PROGRAM MOVMENT_Controller
VAR
	X_Axis:				FB_PTP_AXIS_ABS_CONTROL;
	Y_Axis:				FB_PTP_AXIS_ABS_CONTROL;
	Z_Axis:				FB_PTP_AXIS_ABS_CONTROL;
	
	eJogMode: 				E_JogMode;
END_VAR

IF (G_sControl.ManualMoveMode) THEN
	eJogMode:= MC_JOGMODE_CONTINOUS;
ELSE
	eJogMode:= MC_JOGMODE_INCHING;
END_IF

ACT_AXIS_CTRL();

ACTION ACT_AXIS_CTRL:
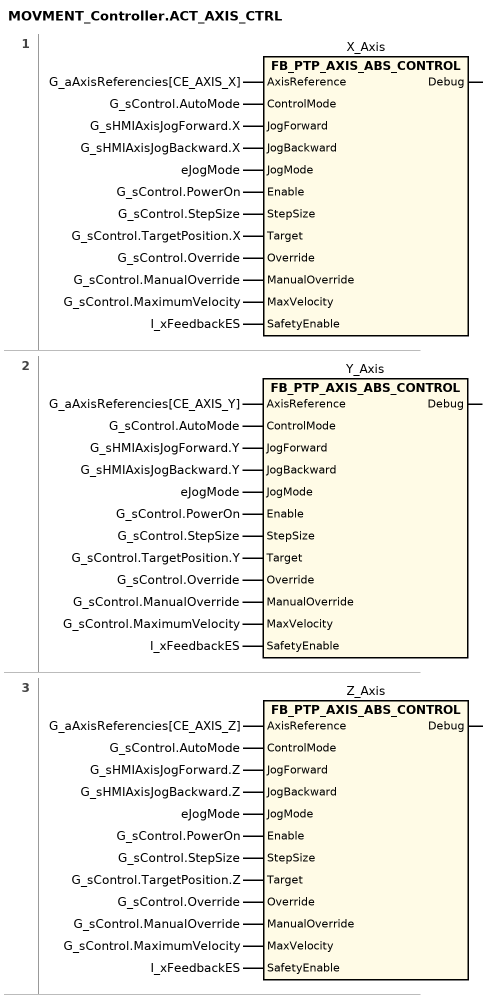
// NETWORK 1
X_Axis(
    AxisReference := G_aAxisReferencies[CE_AXIS_X],
    ControlMode := G_sControl.AutoMode,
    JogForward := G_sHMIAxisJogForward.X,
    JogBackward := G_sHMIAxisJogBackward.X,
    JogMode := eJogMode,
    Enable := G_sControl.PowerOn,
    StepSize := G_sControl.StepSize,
    Target := G_sControl.TargetPosition.X,
    Override := G_sControl.Override,
    ManualOverride := G_sControl.ManualOverride,
    MaxVelocity := G_sControl.MaximumVelocity,
    SafetyEnable := I_xFeedbackES); // FB_PTP_AXIS_ABS_CONTROL

// NETWORK 2
Y_Axis(
    AxisReference := G_aAxisReferencies[CE_AXIS_Y],
    ControlMode := G_sControl.AutoMode,
    JogForward := G_sHMIAxisJogForward.Y,
    JogBackward := G_sHMIAxisJogBackward.Y,
    JogMode := eJogMode,
    Enable := G_sControl.PowerOn,
    StepSize := G_sControl.StepSize,
    Target := G_sControl.TargetPosition.Y,
    Override := G_sControl.Override,
    ManualOverride := G_sControl.ManualOverride,
    MaxVelocity := G_sControl.MaximumVelocity,
    SafetyEnable := I_xFeedbackES); // FB_PTP_AXIS_ABS_CONTROL

// NETWORK 3
Z_Axis(
    AxisReference := G_aAxisReferencies[CE_AXIS_Z],
    ControlMode := G_sControl.AutoMode,
    JogForward := G_sHMIAxisJogForward.Z,
    JogBackward := G_sHMIAxisJogBackward.Z,
    JogMode := eJogMode,
    Enable := G_sControl.PowerOn,
    StepSize := G_sControl.StepSize,
    Target := G_sControl.TargetPosition.Z,
    Override := G_sControl.Override,
    ManualOverride := G_sControl.ManualOverride,
    MaxVelocity := G_sControl.MaximumVelocity,
    SafetyEnable := I_xFeedbackES); // FB_PTP_AXIS_ABS_CONTROL
END_ACTION

END_PROGRAM

(* stored: Version 1.1.0.1, ProductVersion 3.1.4022.18
   POU MOVMENT_Controller: Id {a2fe314f-6d1e-4f60-ac7b-21079c309df6}, SpecialFunc None
   Action ACT_AXIS_CTRL: Id {502e52c1-8be0-4a14-981f-660483023440} *)
